ABB RAPID module: Module1.mod

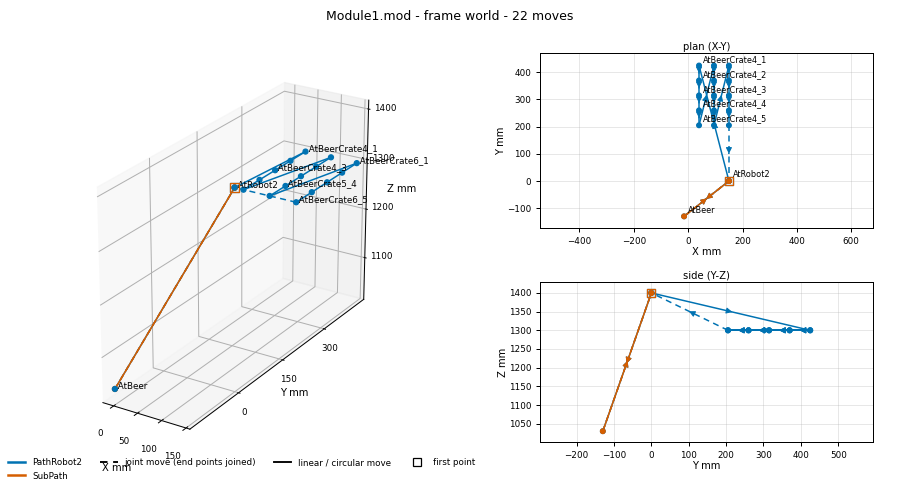
[picture p0: tool path of Module1.mod in frame world, 22 of 22 moves have a stored position in this frame; points joined in program order, loops and branches not executed]
MODULE Module1
	CONST robtarget AtRobot2:=[[150,0,1400],[0,1,0,0],[0,0,0,0],[9E+09,9E+09,9E+09,9E+09,9E+09,9E+09]];
	CONST robtarget AtBeer:=[[-15,-130,1030],[0,1,0,0],[0,0,0,0],[9E+09,9E+09,9E+09,9E+09,9E+09,9E+09]];
	CONST robtarget AtBeerCrate4_1:=[[40,425,1300],[0,1,0,0],[-1,0,-1,0],[9E+09,9E+09,9E+09,9E+09,9E+09,9E+09]];
	CONST robtarget AtBeerCrate4_2:=[[40,370,1300],[0,1,0,0],[-1,0,-1,0],[9E+09,9E+09,9E+09,9E+09,9E+09,9E+09]];
	CONST robtarget AtBeerCrate4_3:=[[40,315,1300],[0,1,0,0],[-1,0,-1,0],[9E+09,9E+09,9E+09,9E+09,9E+09,9E+09]];
	CONST robtarget AtBeerCrate4_4:=[[40,260,1300],[0,1,0,0],[-1,0,-1,0],[9E+09,9E+09,9E+09,9E+09,9E+09,9E+09]];
	CONST robtarget AtBeerCrate4_5:=[[40,205,1300],[0,1,0,0],[-1,0,-1,0],[9E+09,9E+09,9E+09,9E+09,9E+09,9E+09]];
	CONST robtarget AtBeerCrate5_1:=[[95,425,1300],[0,1,0,0],[-1,0,-1,0],[9E+09,9E+09,9E+09,9E+09,9E+09,9E+09]];
	CONST robtarget AtBeerCrate5_2:=[[95,370,1300],[0,1,0,0],[-1,0,-1,0],[9E+09,9E+09,9E+09,9E+09,9E+09,9E+09]];
	CONST robtarget AtBeerCrate5_3:=[[95,315,1300],[0,1,0,0],[-1,0,-1,0],[9E+09,9E+09,9E+09,9E+09,9E+09,9E+09]];
	CONST robtarget AtBeerCrate5_4:=[[95,260,1300],[0,1,0,0],[-1,0,-1,0],[9E+09,9E+09,9E+09,9E+09,9E+09,9E+09]];
	CONST robtarget AtBeerCrate5_5:=[[95,205,1300],[0,1,0,0],[0,0,0,0],[9E+09,9E+09,9E+09,9E+09,9E+09,9E+09]];
	CONST robtarget AtBeerCrate6_1:=[[150,425,1300],[0,1,0,0],[0,0,0,0],[9E+09,9E+09,9E+09,9E+09,9E+09,9E+09]];
	CONST robtarget AtBeerCrate6_2:=[[150,370,1300],[0,1,0,0],[0,0,0,0],[9E+09,9E+09,9E+09,9E+09,9E+09,9E+09]];
	CONST robtarget AtBeerCrate6_3:=[[150,315,1300],[0,1,0,0],[0,0,0,0],[9E+09,9E+09,9E+09,9E+09,9E+09,9E+09]];
	CONST robtarget AtBeerCrate6_4:=[[150,260,1300],[0,1,0,0],[0,0,0,0],[9E+09,9E+09,9E+09,9E+09,9E+09,9E+09]];
	CONST robtarget AtBeerCrate6_5:=[[150,205,1300],[0,1,0,0],[0,0,0,0],[9E+09,9E+09,9E+09,9E+09,9E+09,9E+09]];
    !***********************************************************
    !
    ! Module:  Module1
    !
    ! Description:
    !   <Insert description here>
    !
    ! Author: Bruger
    !
    ! Version: 1.0
    !
    !***********************************************************


    !***********************************************************
    !
    ! Procedure main
    !
    !   This is the entry point of your program
    !
    !***********************************************************
    PROC main()
		PathRobot2;
        !Add your code here
    ENDPROC
	PROC PathRobot2()
	    MoveJ AtRobot2,v2000,z100,Tool2\WObj:=wobj0;
	    WaitDI Di1CrateReadyForFilling,1;
	    WaitTime 1.5;
	    MoveL AtBeer,v2000,fine,Tool2\WObj:=wobj0;
	    SetDO Do2Gripper,0;
	    WaitTime 0.3;
	    MoveJ AtRobot2,v2000,z100,Tool2\WObj:=wobj0;
	    MoveL AtBeerCrate4_1,v2000,fine,Tool2\WObj:=wobj0;
	    SubPath;
	    MoveL AtBeerCrate4_2,v2000,fine,Tool2\WObj:=wobj0;
	    SubPath;
	    MoveL AtBeerCrate4_3,v2000,fine,Tool2\WObj:=wobj0;
	    SubPath;
	    MoveL AtBeerCrate4_4,v2000,fine,Tool2\WObj:=wobj0;
	    SubPath;
	    MoveL AtBeerCrate4_5,v2000,fine,Tool2\WObj:=wobj0;
	    SubPath;
	    MoveL AtBeerCrate5_1,v2000,fine,Tool2\WObj:=wobj0;
	    SubPath;
	    MoveL AtBeerCrate5_2,v2000,fine,Tool2\WObj:=wobj0;
	    SubPath;
	    MoveL AtBeerCrate5_3,v2000,fine,Tool2\WObj:=wobj0;
	    SubPath;
	    MoveL AtBeerCrate5_4,v2000,fine,Tool2\WObj:=wobj0;
	    SubPath;
	    MoveL AtBeerCrate5_5,v2000,fine,Tool2\WObj:=wobj0;
	    SubPath;
	    MoveL AtBeerCrate6_1,v2000,fine,Tool2\WObj:=wobj0;
	    SubPath;
	    MoveL AtBeerCrate6_2,v2000,fine,Tool2\WObj:=wobj0;
	    SubPath;
	    MoveL AtBeerCrate6_3,v2000,fine,Tool2\WObj:=wobj0;
	    SubPath;
	    MoveL AtBeerCrate6_4,v2000,fine,Tool2\WObj:=wobj0;
	    SubPath;
	    MoveL AtBeerCrate6_5,v2000,fine,Tool2\WObj:=wobj0;
	    SetDO Do2Gripper,0;
		WaitTime 0.3;
		MoveJ AtRobot2,v2000,z100,Tool2\WObj:=wobj0;
	ENDPROC
	PROC SubPath()
	    SetDO Do2Gripper,0;
	    WaitTime 0.3;
	    MoveJ AtRobot2,v2000,z100,Tool2\WObj:=wobj0;
	    MoveL AtBeer,v2000,fine,Tool2\WObj:=wobj0;
	    SetDO Do2Gripper,1;
	    WaitTime 0.3;
	    MoveJ AtRobot2,v2000,z100,Tool2\WObj:=wobj0;
	ENDPROC
ENDMODULE
